FUNCTION_BLOCK FB_CommandChangeComplete EXTENDS FB_CommandChange  IMPLEMENTS ITF_CommandChange
VAR

END_VAR

METHOD Execute : BOOL
VAR_INPUT
END_VAR
END_METHOD

METHOD FB_init : BOOL
VAR_INPUT
	bInitRetains : BOOL; // if TRUE, the retain variables are initialized (warm start / cold start)
	bInCopyCode : BOOL;  // if TRUE, the instance afterwards gets moved into the copy code (online change)
END_VAR
THIS^.SetText (eLocation := E_BaseLocation.pl, wsDescription := "Command change state - Complete");
THIS^.SetText (eLocation := E_BaseLocation.en, wsDescription := "Command change state - Complete");
THIS^.SetText (eLocation := E_BaseLocation.de, wsDescription := "Command change state - Complete");
THIS^.SetName (stName := THIS^.GetTexts ());
END_METHOD

END_FUNCTION_BLOCK

(* stored: Version 1.1.0.1
   POU FB_CommandChangeComplete: Id {64939450-2f92-0c92-20b1-eaf3248da179}, SpecialFunc None
   Method Execute: Id {c278a172-f4b6-080b-0c34-b72bb9a46919}
   Method FB_init: Id {4dd750f3-15c9-0c87-3fb8-51fc75b2803d} *)
